SYSTEM LIFTER_MVL (* Lifter with Feed & Takeoff Conveyors *)
  (* Standard: 61499-1; Classification: Simulation; ApplicationDomain: Assembly; Type: Dual Stroke Cylinder *)
  (* Version 0.4, 2007-07-08, JHC, Holobloc Inc, Changed MODEL.UI.FAULT,CLOCK.FAULT  to SUBL_0; added MODEL.CLOCK.CLK_DLY. *)
  (* Version 0.3, 2004-12-19, JHC, Rockwell Automation, Adjusted frame heights for WinXP. *)
  (* Version 0.2, 2004-11-11, JHC, Rockwell Automation, Combined XFER_MDL, FAULT_MDL; added faults from UIs. *)
  (* Version 0.1, 2004-10-29, JHC, Rockwell Automation, Changed FEED_MDL.FEED to CNVG_MDLL. *)
  (* Version 0.0, 2004-09-29, JHC, Rockwell Automation, Extended from LIFTER_VIEWL. *)
  DEVICE HMI : FRAME_DEVICE(BOUNDS := [100,100,325,195], GRID := [3,2])
    RESOURCE TAKEOFF_SENSORS : PANEL_RESOURCE
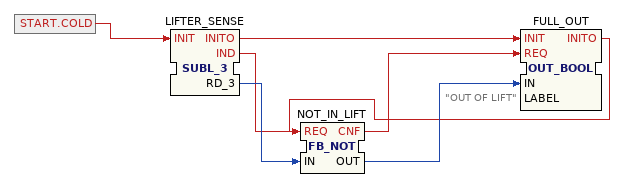
      FBS
        LIFTER_SENSE : SUBL_3;
        FULL_OUT : OUT_BOOL(LABEL := "OUT OF LIFT");
        NOT_IN_LIFT : FB_NOT;
      END_FBS
      EVENT_CONNECTIONS
        START.COLD TO LIFTER_SENSE.INIT;
        LIFTER_SENSE.INITO TO FULL_OUT.INIT;
        LIFTER_SENSE.IND TO NOT_IN_LIFT.REQ;
        NOT_IN_LIFT.CNF TO FULL_OUT.REQ;
        FULL_OUT.INITO TO NOT_IN_LIFT.REQ;
      END_CONNECTIONS
      DATA_CONNECTIONS
        LIFTER_SENSE.RD_3 TO NOT_IN_LIFT.IN;
        NOT_IN_LIFT.OUT TO FULL_OUT.IN;
      END_CONNECTIONS
    END_RESOURCE
    RESOURCE TAKEOFF_ACTUATORS : PANEL_RESOURCE
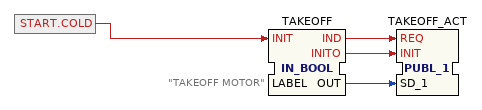
      FBS
        TAKEOFF : IN_BOOL(LABEL := "TAKEOFF MOTOR");
        TAKEOFF_ACT : PUBL_1;
      END_FBS
      EVENT_CONNECTIONS
        START.COLD TO TAKEOFF.INIT;
        TAKEOFF.IND TO TAKEOFF_ACT.REQ;
        TAKEOFF.INITO TO TAKEOFF_ACT.INIT;
      END_CONNECTIONS
      DATA_CONNECTIONS
        TAKEOFF.OUT TO TAKEOFF_ACT.SD_1;
      END_CONNECTIONS
    END_RESOURCE
    RESOURCE LIFT_SENSORS : PANEL_RESOURCE(ROWS := 2, COLS := 2)
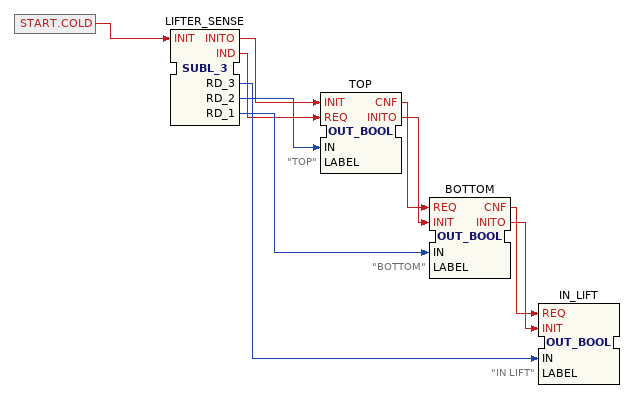
      FBS
        LIFTER_SENSE : SUBL_3;
        IN_LIFT : OUT_BOOL(LABEL := "IN LIFT");
        TOP : OUT_BOOL(LABEL := "TOP");
        BOTTOM : OUT_BOOL(LABEL := "BOTTOM");
      END_FBS
      EVENT_CONNECTIONS
        START.COLD TO LIFTER_SENSE.INIT;
        TOP.CNF TO BOTTOM.REQ;
        TOP.INITO TO BOTTOM.INIT;
        LIFTER_SENSE.INITO TO TOP.INIT;
        LIFTER_SENSE.IND TO TOP.REQ;
        BOTTOM.CNF TO IN_LIFT.REQ;
        BOTTOM.INITO TO IN_LIFT.INIT;
      END_CONNECTIONS
      DATA_CONNECTIONS
        LIFTER_SENSE.RD_3 TO IN_LIFT.IN;
        LIFTER_SENSE.RD_2 TO TOP.IN;
        LIFTER_SENSE.RD_1 TO BOTTOM.IN;
      END_CONNECTIONS
    END_RESOURCE
    RESOURCE LIFT_ACTUATORS : PANEL_RESOURCE(ROWS := 2, COLS := 2)
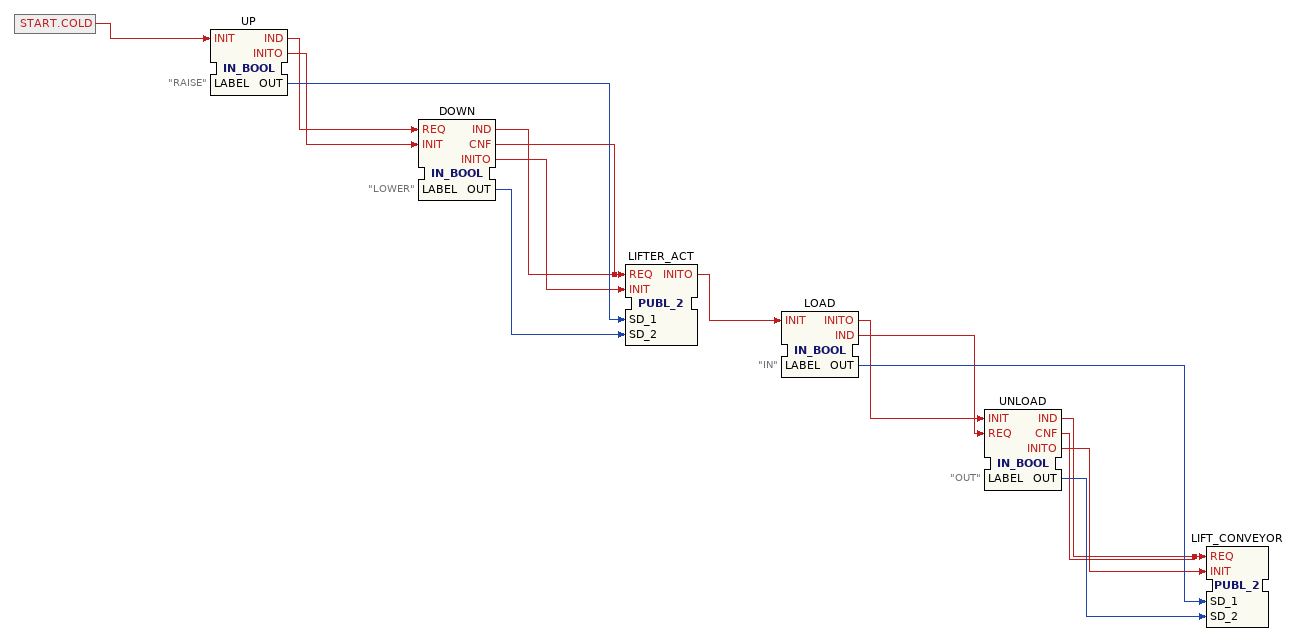
      FBS
        UP : IN_BOOL(LABEL := "RAISE");
        LIFTER_ACT : PUBL_2;
        DOWN : IN_BOOL(LABEL := "LOWER");
        LOAD : IN_BOOL(LABEL := "IN");
        UNLOAD : IN_BOOL(LABEL := "OUT");
        LIFT_CONVEYOR : PUBL_2;
      END_FBS
      EVENT_CONNECTIONS
        START.COLD TO UP.INIT;
        LOAD.INITO TO UNLOAD.INIT;
        LOAD.IND TO UNLOAD.REQ;
        DOWN.IND TO LIFTER_ACT.REQ;
        UP.IND TO DOWN.REQ;
        DOWN.CNF TO LIFTER_ACT.REQ;
        UP.INITO TO DOWN.INIT;
        UNLOAD.IND TO LIFT_CONVEYOR.REQ;
        UNLOAD.CNF TO LIFT_CONVEYOR.REQ;
        DOWN.INITO TO LIFTER_ACT.INIT;
        LIFTER_ACT.INITO TO LOAD.INIT;
        UNLOAD.INITO TO LIFT_CONVEYOR.INIT;
      END_CONNECTIONS
      DATA_CONNECTIONS
        LOAD.OUT TO LIFT_CONVEYOR.SD_1;
        UNLOAD.OUT TO LIFT_CONVEYOR.SD_2;
        UP.OUT TO LIFTER_ACT.SD_1;
        DOWN.OUT TO LIFTER_ACT.SD_2;
      END_CONNECTIONS
    END_RESOURCE
    RESOURCE FEED_SENSORS : PANEL_RESOURCE
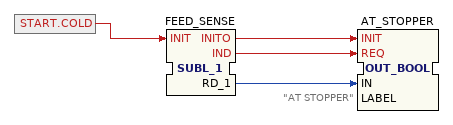
      FBS
        FEED_SENSE : SUBL_1;
        AT_STOPPER : OUT_BOOL(LABEL := "AT STOPPER");
      END_FBS
      EVENT_CONNECTIONS
        START.COLD TO FEED_SENSE.INIT;
        FEED_SENSE.INITO TO AT_STOPPER.INIT;
        FEED_SENSE.IND TO AT_STOPPER.REQ;
      END_CONNECTIONS
      DATA_CONNECTIONS
        FEED_SENSE.RD_1 TO AT_STOPPER.IN;
      END_CONNECTIONS
    END_RESOURCE
    RESOURCE FEED_ACTUATORS : PANEL_RESOURCE
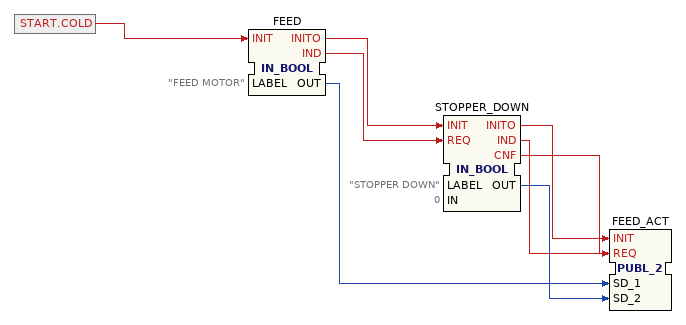
      FBS
        FEED : IN_BOOL(LABEL := "FEED MOTOR");
        FEED_ACT : PUBL_2;
        STOPPER_DOWN : IN_BOOL(LABEL := "STOPPER DOWN", IN := 0);
      END_FBS
      EVENT_CONNECTIONS
        FEED.INITO TO STOPPER_DOWN.INIT;
        FEED.IND TO STOPPER_DOWN.REQ;
        START.COLD TO FEED.INIT;
        STOPPER_DOWN.INITO TO FEED_ACT.INIT;
        STOPPER_DOWN.IND TO FEED_ACT.REQ;
        STOPPER_DOWN.CNF TO FEED_ACT.REQ;
      END_CONNECTIONS
      DATA_CONNECTIONS
        FEED.OUT TO FEED_ACT.SD_1;
        STOPPER_DOWN.OUT TO FEED_ACT.SD_2;
      END_CONNECTIONS
    END_RESOURCE
  END_DEVICE
  DEVICE MODEL : FRAME_DEVICE(BOUNDS := [425,100,160,260])
    RESOURCE CLOCK : EMB_RES
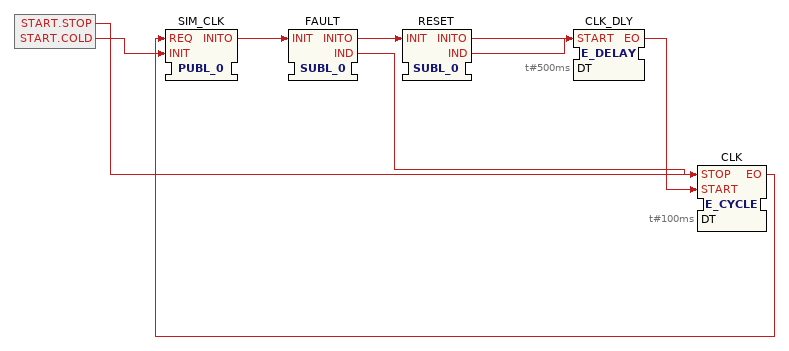
      FBS
        CLK : E_CYCLE(DT := t#100ms);
        SIM_CLK : PUBL_0;
        FAULT : SUBL_0;
        RESET : SUBL_0;
        CLK_DLY : E_DELAY(DT := t#500ms);
      END_FBS
      EVENT_CONNECTIONS
        START.STOP TO CLK.STOP;
        CLK.EO TO SIM_CLK.REQ;
        START.COLD TO SIM_CLK.INIT;
        SIM_CLK.INITO TO FAULT.INIT;
        FAULT.INITO TO RESET.INIT;
        FAULT.IND TO CLK.STOP;
        RESET.INITO TO CLK_DLY.START;
        RESET.IND TO CLK_DLY.START;
        CLK_DLY.EO TO CLK.START;
      END_CONNECTIONS
    END_RESOURCE
    RESOURCE FEED_MDL : EMB_RES
      FBS
        FEED : CNVG_MDLL(VF := 20, VS := 50);
        FEED_UNLD : SUBL_0;
        RESET : SUBL_0;
        WARN : SUBL_2;
        WARNING : LOADLE(LPOS := 100, STYLE := VSTYLE#PALLET, WKPC := [255,255,0], ID := "FEED_LOAD");
        JAM_OR_HALFIN : FB_OR;
        FAULT : SUBL_2;
        CRUSHED : E_PERMIT;
        DROPPED : LOADLE(ID := "FEED_LOAD", LPOS := 100, STYLE := VSTYLE#PALLET, WKPC := [255,0,0]);
      END_FBS
      EVENT_CONNECTIONS
        START.COLD TO FEED.INIT;
        FEED.INITO TO FEED_UNLD.INIT;
        FEED_UNLD.INITO TO RESET.INIT;
        RESET.IND TO FEED.UNLD;
        RESET.INITO TO WARN.INIT;
        WARN.IND TO JAM_OR_HALFIN.REQ;
        START.COLD TO FAULT.INIT;
        WARN.INITO TO WARNING.INIT;
        JAM_OR_HALFIN.CNF TO WARNING.REQ;
        FAULT.IND TO CRUSHED.EI;
        CRUSHED.EO TO FEED.UNLD;
        FAULT.IND TO DROPPED.REQ;
        WARNING.INITO TO DROPPED.INIT;
        FEED_UNLD.IND TO FEED.UNLD;
      END_CONNECTIONS
      DATA_CONNECTIONS
        WARN.RD_1 TO JAM_OR_HALFIN.IN1;
        WARN.RD_2 TO JAM_OR_HALFIN.IN2;
        JAM_OR_HALFIN.OUT TO WARNING.QI;
        FAULT.RD_1 TO CRUSHED.PERMIT;
        FAULT.RD_2 TO DROPPED.QI;
      END_CONNECTIONS
    END_RESOURCE
    RESOURCE LIFTER_MDL : EMB_RES
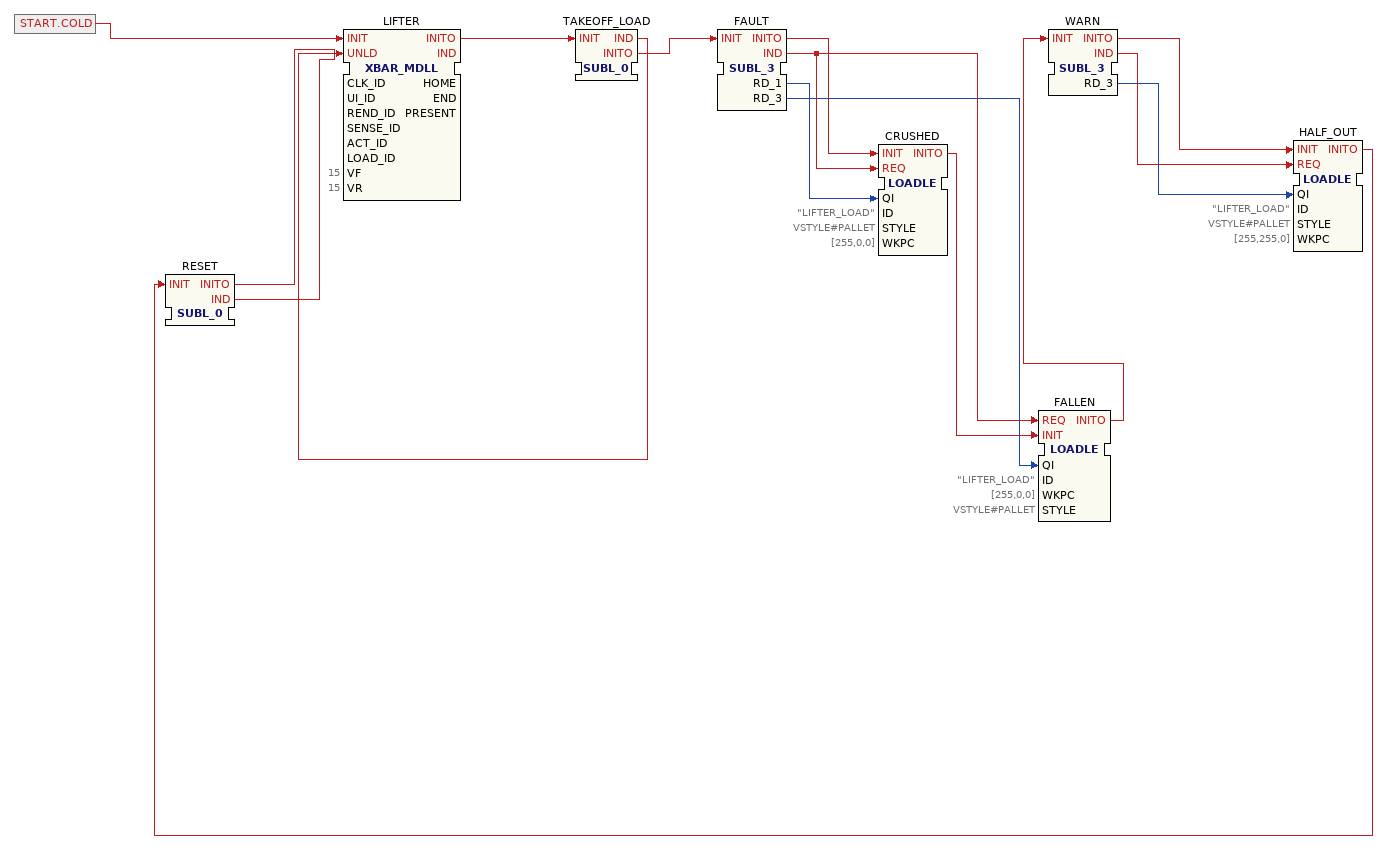
      FBS
        LIFTER : XBAR_MDLL(VF := 15, VR := 15);
        TAKEOFF_LOAD : SUBL_0;
        FAULT : SUBL_3;
        CRUSHED : LOADLE(ID := "LIFTER_LOAD", STYLE := VSTYLE#PALLET, WKPC := [255,0,0]);
        FALLEN : LOADLE(ID := "LIFTER_LOAD", WKPC := [255,0,0], STYLE := VSTYLE#PALLET);
        RESET : SUBL_0;
        WARN : SUBL_3;
        HALF_OUT : LOADLE(ID := "LIFTER_LOAD", STYLE := VSTYLE#PALLET, WKPC := [255,255,0]);
      END_FBS
      EVENT_CONNECTIONS
        START.COLD TO LIFTER.INIT;
        LIFTER.INITO TO TAKEOFF_LOAD.INIT;
        TAKEOFF_LOAD.IND TO LIFTER.UNLD;
        TAKEOFF_LOAD.INITO TO FAULT.INIT;
        FAULT.INITO TO CRUSHED.INIT;
        FAULT.IND TO CRUSHED.REQ;
        FAULT.IND TO FALLEN.REQ;
        CRUSHED.INITO TO FALLEN.INIT;
        WARN.INITO TO HALF_OUT.INIT;
        WARN.IND TO HALF_OUT.REQ;
        RESET.INITO TO LIFTER.UNLD;
        RESET.IND TO LIFTER.UNLD;
        FALLEN.INITO TO WARN.INIT;
        HALF_OUT.INITO TO RESET.INIT;
      END_CONNECTIONS
      DATA_CONNECTIONS
        FAULT.RD_1 TO CRUSHED.QI;
        FAULT.RD_3 TO FALLEN.QI;
        WARN.RD_3 TO HALF_OUT.QI;
      END_CONNECTIONS
    END_RESOURCE
    RESOURCE XFER_MDL : EMB_RES (* Pallet Transfer Model *)
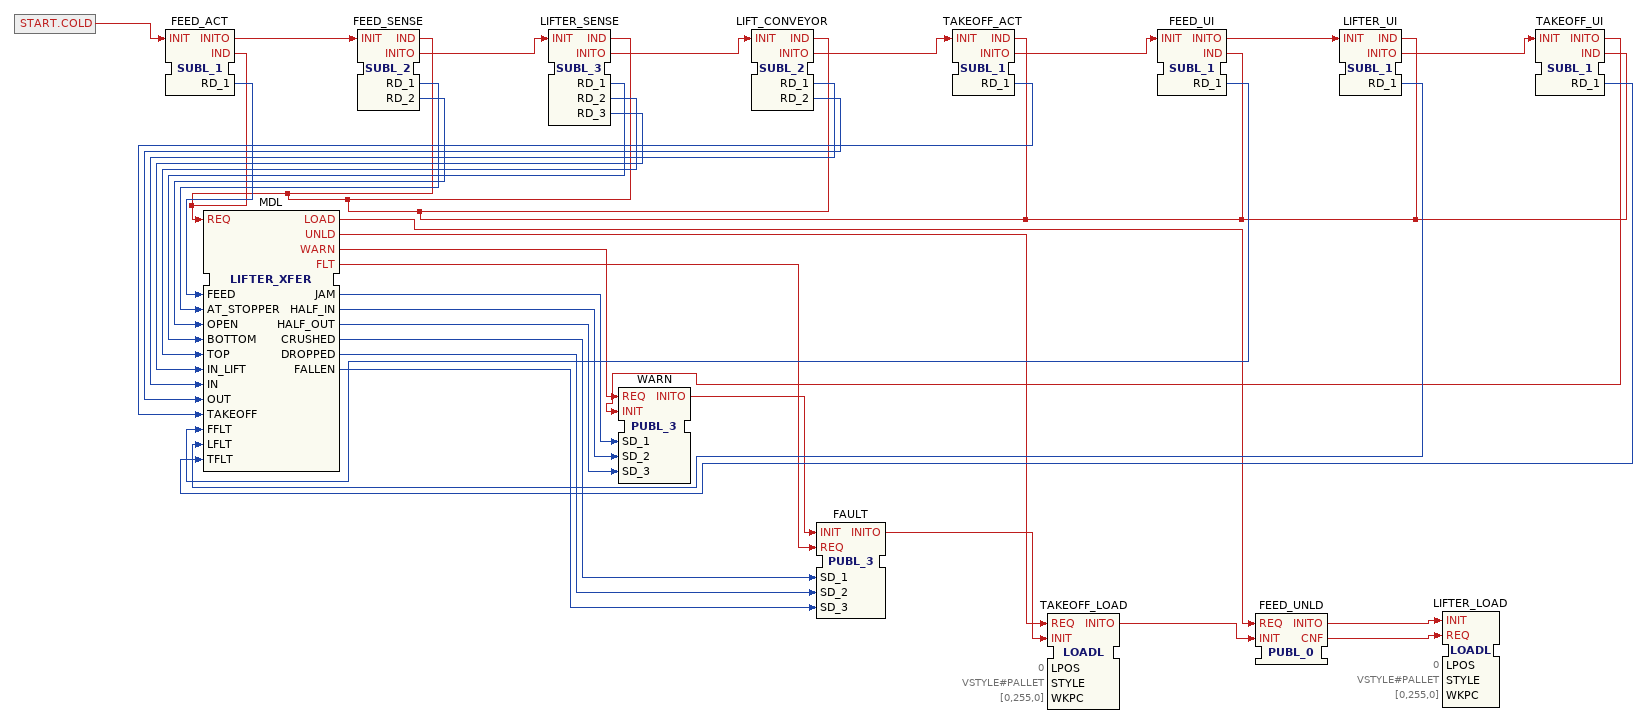
      FBS
        MDL : LIFTER_XFER;
        FEED_ACT : SUBL_1;
        FEED_SENSE : SUBL_2;
        LIFTER_SENSE : SUBL_3;
        LIFT_CONVEYOR : SUBL_2;
        TAKEOFF_ACT : SUBL_1;
        LIFTER_LOAD : LOADL(LPOS := 0, STYLE := VSTYLE#PALLET, WKPC := [0,255,0]);
        TAKEOFF_LOAD : LOADL(LPOS := 0, STYLE := VSTYLE#PALLET, WKPC := [0,255,0]);
        LIFTER_UI : SUBL_1;
        WARN : PUBL_3;
        FAULT : PUBL_3;
        FEED_UNLD : PUBL_0;
        FEED_UI : SUBL_1;
        TAKEOFF_UI : SUBL_1;
      END_FBS
      EVENT_CONNECTIONS
        START.COLD TO FEED_ACT.INIT;
        FEED_ACT.INITO TO FEED_SENSE.INIT;
        FEED_ACT.IND TO MDL.REQ;
        FEED_SENSE.IND TO MDL.REQ;
        FEED_SENSE.INITO TO LIFTER_SENSE.INIT;
        LIFTER_SENSE.IND TO MDL.REQ;
        LIFTER_SENSE.INITO TO LIFT_CONVEYOR.INIT;
        LIFT_CONVEYOR.IND TO MDL.REQ;
        LIFT_CONVEYOR.INITO TO TAKEOFF_ACT.INIT;
        TAKEOFF_ACT.IND TO MDL.REQ;
        LIFTER_UI.IND TO MDL.REQ;
        MDL.UNLD TO TAKEOFF_LOAD.REQ;
        WARN.INITO TO FAULT.INIT;
        MDL.WARN TO WARN.REQ;
        MDL.FLT TO FAULT.REQ;
        FAULT.INITO TO TAKEOFF_LOAD.INIT;
        MDL.LOAD TO FEED_UNLD.REQ;
        FEED_UNLD.INITO TO LIFTER_LOAD.INIT;
        FEED_UNLD.CNF TO LIFTER_LOAD.REQ;
        TAKEOFF_LOAD.INITO TO FEED_UNLD.INIT;
        TAKEOFF_ACT.INITO TO FEED_UI.INIT;
        FEED_UI.INITO TO LIFTER_UI.INIT;
        LIFTER_UI.INITO TO TAKEOFF_UI.INIT;
        TAKEOFF_UI.INITO TO WARN.INIT;
        FEED_UI.IND TO MDL.REQ;
        TAKEOFF_UI.IND TO MDL.REQ;
      END_CONNECTIONS
      DATA_CONNECTIONS
        FEED_ACT.RD_1 TO MDL.FEED;
        FEED_SENSE.RD_1 TO MDL.AT_STOPPER;
        LIFTER_SENSE.RD_1 TO MDL.BOTTOM;
        LIFTER_SENSE.RD_2 TO MDL.TOP;
        LIFTER_SENSE.RD_3 TO MDL.IN_LIFT;
        LIFT_CONVEYOR.RD_1 TO MDL.IN;
        LIFT_CONVEYOR.RD_2 TO MDL.OUT;
        TAKEOFF_ACT.RD_1 TO MDL.TAKEOFF;
        FEED_SENSE.RD_2 TO MDL.OPEN;
        LIFTER_UI.RD_1 TO MDL.LFLT;
        MDL.JAM TO WARN.SD_1;
        MDL.HALF_IN TO WARN.SD_2;
        MDL.HALF_OUT TO WARN.SD_3;
        MDL.CRUSHED TO FAULT.SD_1;
        MDL.DROPPED TO FAULT.SD_2;
        MDL.FALLEN TO FAULT.SD_3;
        FEED_UI.RD_1 TO MDL.FFLT;
        TAKEOFF_UI.RD_1 TO MDL.TFLT;
      END_CONNECTIONS
    END_RESOURCE
    RESOURCE TAKEOFF_MDL : EMB_RES
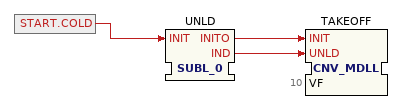
      FBS
        TAKEOFF : CNV_MDLL(VF := 10);
        UNLD : SUBL_0;
      END_FBS
      EVENT_CONNECTIONS
        START.COLD TO UNLD.INIT;
        UNLD.INITO TO TAKEOFF.INIT;
        UNLD.IND TO TAKEOFF.UNLD;
      END_CONNECTIONS
    END_RESOURCE
    RESOURCE UI : PANEL_RESOURCE(ROWS := 2, COLS := 2)
      FBS
        FAULT_IND : OUT_BOOL(LABEL := "FAULT ", C1 := [255,0,0]);
        RESET_PB : IN_EVENT(LABEL := "RESET");
        RESET : PUBL_0;
        LOAD_PB : IN_EVENT(LABEL := "LOAD");
        UNLD_PB : IN_EVENT(LABEL := "UNLOAD");
        FEED_LOAD : LOADL(STYLE := VSTYLE#PALLET, WKPC := [0,255,0]);
        UNLD : PUBL_0;
        FLT : E_RS;
        FAULT : SUBL_0;
      END_FBS
      EVENT_CONNECTIONS
        FAULT_IND.INITO TO RESET_PB.INIT;
        RESET_PB.INITO TO RESET.INIT;
        RESET_PB.IND TO RESET.REQ;
        START.COLD TO LOAD_PB.INIT;
        LOAD_PB.INITO TO FEED_LOAD.INIT;
        FEED_LOAD.INITO TO UNLD_PB.INIT;
        LOAD_PB.IND TO FEED_LOAD.REQ;
        UNLD_PB.INITO TO UNLD.INIT;
        UNLD_PB.IND TO UNLD.REQ;
        UNLD.INITO TO FAULT_IND.INIT;
        RESET.CNF TO UNLD.REQ;
        FLT.EO TO FAULT_IND.REQ;
        RESET.INITO TO FAULT.INIT;
        FAULT.IND TO FLT.S;
        UNLD.CNF TO FLT.R;
      END_CONNECTIONS
      DATA_CONNECTIONS
        FLT.Q TO FAULT_IND.IN;
      END_CONNECTIONS
    END_RESOURCE
    RESOURCE VIEW : VIEW_PANEL(DIA := 30, SIZE := [5,5], VERTICAL := 1)
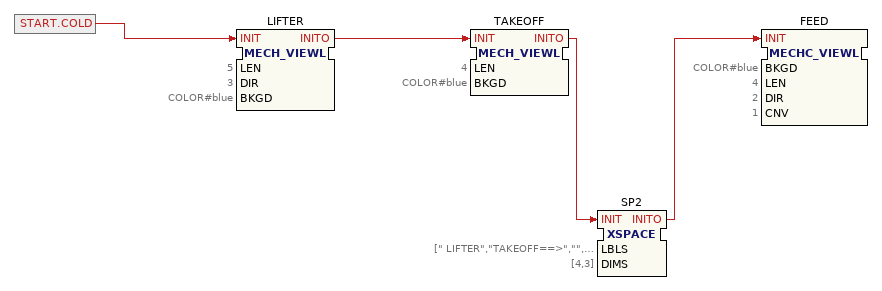
      FBS
        LIFTER : MECH_VIEWL(LEN := 5, DIR := 3, BKGD := COLOR#blue);
        FEED : MECHC_VIEWL(BKGD := COLOR#blue, LEN := 4, DIR := 2, CNV := 1); (* Feed Conveyor *)
        SP2 : XSPACE(LBLS := [" LIFTER","TAKEOFF==>","","<==FEED"], DIMS := [4,3]);
        TAKEOFF : MECH_VIEWL(LEN := 4, BKGD := COLOR#blue); (* Takeoff Conveyor *)
      END_FBS
      EVENT_CONNECTIONS
        TAKEOFF.INITO TO SP2.INIT;
        SP2.INITO TO FEED.INIT;
        START.COLD TO LIFTER.INIT;
        LIFTER.INITO TO TAKEOFF.INIT;
      END_CONNECTIONS
    END_RESOURCE
  END_DEVICE
END_SYSTEM
